FUNCTION_BLOCK NodeProperty
VAR
	nodeProperty : Property_ANY('','',0);
END_VAR

PROPERTY PUBLIC DataSize : UDINT
GET
DataSize := nodeProperty.DataSize;
END_GET
END_PROPERTY

METHOD FB_init : BOOL
VAR_INPUT
	bInitRetains : BOOL; // if TRUE, the retain variables are initialized (warm start / cold start)
	bInCopyCode : BOOL;  // if TRUE, the instance afterwards gets moved into the copy code (online change)
	Name : STRING;
	DataType : T_MAXSTRING;
	Parent : I_Node;
END_VAR
VAR
	ParentWithProperties : I_HaveProperties;
END_VAR
IF __QUERYINTERFACE(Parent, ParentWithProperties) THEN
	nodeProperty.FB_init(FALSE,FALSE,Name,DataType,ParentWithProperties);
END_IF
END_METHOD

METHOD PUBLIC Get
VAR_INPUT
	Value : ANY;
END_VAR
nodeProperty.Get(Value);
END_METHOD

PROPERTY PUBLIC Name : STRING
GET
Name := nodeProperty.Name;
END_GET
END_PROPERTY

END_FUNCTION_BLOCK

(* stored: Version 1.1.0.1, ProductVersion 3.1.4024.12
   POU NodeProperty: Id {2f3818ec-5c85-0aeb-0525-1e3645adde0b}, SpecialFunc None
   Folder Constructor: Id {df8a62d6-1721-0d78-1a3f-56c93a4a9a60}
   Property DataSize: Id {8e26e426-bbb6-0fbf-0430-5092d76fdbda}
   Get Get: Id {0cd040a5-e36b-0c4d-2416-2d894abf6941}
   Method FB_init: Id {e1fde59c-45aa-0e76-3869-41613069cdff}
   Method Get: Id {442b5a48-b87e-04e7-3785-b0a07f9159e4}
   Property Name: Id {55d2d9df-bcc5-0c95-02c1-bb449c0b3a39}
   Get Get: Id {8b691aa0-20d5-048c-11ba-8a9ae7296964} *)
